(****************************************************************************************)
(*							Beckhoff Automation Poland									*)
(*								F_2ndByteWtoB v1.0										*)
(*									15.02.2010											*)
(*		Funkcja wyciagajaca bardziej znaczacy BYTE ze zmiennej typu WORD				*)
(*							 	wyjscie typu BYTE										*)
(*______________________________________________________________________________________*)
FUNCTION F_2ndByteWtoB : BYTE
VAR_INPUT
	wIn		:	WORD;
END_VAR

F_2ndByteWtoB := WORD_TO_BYTE(SHR(wIn,8));

END_FUNCTION

(* stored: Version 1.1.0.1, ProductVersion 3.1.4026.13, FileIdentifier c434750233ba15be5901e6832bc73bab6380feb6, FileSignature 01b83cdd0ea7e544133b8b642daf23cd6284ed5258314b3ea575f5fa3c97483c89161ff2ba5587ff52b34bbbe5f4d94f4a6c2eb785f866e3b29f902caca511a472053feb55ad435a8e05ee3f27396c8b5aac3af9027a664600261080ed53267062acf8b309dbdb626b5c5224ad11a53d98c25d44311a3bb8ee09d19c3b6ed0b2907a2b73909e6fe4f44963275895ccb1f6d1f12312d5b0501232ecdf5f476db29e914a47e473c16111e534c921a55333efcaab689c01b6d3b5add254f4ed0792fe54a9a898f090a4a35fe7df72e5fff00df6d83ab7d60763e0fb18d8d93b76a21618846c5b29fa7985042286fc9130b8379758e6395652c403cf60c76cf4779b
   POU F_2ndByteWtoB: Id {9e6918ee-b798-4e5c-831c-ebbf6d9329ec}, SpecialFunc None *)
